(* IEC 61131-3 sources: ae-conveyorline/src, 7 files *)

(* ---- ConveyorSimulation.st ---- *)
USING System.Timer;

NAMESPACE Simatic.Ax.Simulation
    /// Simulation class for conveyor sensor signals using shift register approach
    /// Simulates packages moving along 1 conveyor line (3 conveyors total)
    CLASS ConveyorSimulation
        VAR CONSTANT
            CONVEYOR_LENGTH : LREAL := 2.0; // Conveyor length in meters
            CONVEYOR_SPEED : LREAL := 1.5;  // Conveyor speed in m/s
            SHIFT_INTERVAL : TIME := T#100ms; // Time interval for shift register update
            REGISTER_SIZE : INT := 30; // Size of shift register (3 seconds / 100ms = 30 positions)
            PACKAGE_INTERVAL_POSITIONS : INT := 20; // Positions between packages (2s / 100ms = 20)
        END_VAR

        VAR PUBLIC
            /// Enable/disable simulation
            SimulationEnabled : BOOL := FALSE;

            /// Simulated sensor outputs (3 Conveyors)
            Sensor1 : BOOL := FALSE;
            Sensor2 : BOOL := FALSE;
            Sensor3 : BOOL := FALSE;
        END_VAR

        VAR PRIVATE
            // Shift register for the conveyor line
            _shiftRegister : ARRAY[0..29] OF BOOL;

            // Timer for shift register update
            _shiftTimer : OnDelay;
            _shiftTimerReset : BOOL := FALSE;

            // Package generation counter
            _packageCounter : INT := 0;

            // Sensor position mapping (in shift register positions)
            _sensor1Position : INT := 0;   // Position 0 (start)
            _sensor2Position : INT := 10;  // Position 10 (after 1.0s)
            _sensor3Position : INT := 20;  // Position 20 (after 2.0s)

            // Sensor trigger window
            _sensorWindow : INT := 5; // 5 positions = 500ms

            // Initialization flag
            _initialized : BOOL := FALSE;
        END_VAR

        /// Initialize simulation
        METHOD PUBLIC Initialize
            VAR_TEMP
                i : INT;
            END_VAR

            // Clear shift register
            FOR i := 0 TO (REGISTER_SIZE - 1) DO
                _shiftRegister[i] := FALSE;
            END_FOR;

            _packageCounter := 0;
            _initialized := TRUE;
        END_METHOD

        /// Cyclic update method - must be called every PLC cycle
        METHOD PUBLIC Update
            VAR_TEMP
                i : INT;
            END_VAR

            // If simulation is disabled, reset all sensors
            IF NOT SimulationEnabled THEN
                IF _initialized THEN
                    THIS.Initialize();
                    _initialized := FALSE;
                END_IF;
                THIS.ResetAllSensors();
                RETURN;
            END_IF;

            // Initialize on first run
            IF NOT _initialized THEN
                THIS.Initialize();
            END_IF;

            // Update shift register at defined interval
            _shiftTimer(signal := NOT _shiftTimerReset, duration := SHIFT_INTERVAL);

            IF _shiftTimer.output THEN
                // Shift all positions one step forward
                FOR i := (REGISTER_SIZE - 1) TO 1 BY -1 DO
                    _shiftRegister[i] := _shiftRegister[i - 1];
                END_FOR;

                // Generate new packages
                _packageCounter := _packageCounter + 1;
                IF _packageCounter >= PACKAGE_INTERVAL_POSITIONS THEN
                    _shiftRegister[0] := TRUE;
                    _packageCounter := 0;
                ELSE
                    _shiftRegister[0] := FALSE;
                END_IF;

                // Reset timer for next cycle
                _shiftTimerReset := TRUE;
            ELSE
                _shiftTimerReset := FALSE;
            END_IF;

            // Update sensor outputs (3 Conveyors)
            Sensor1 := THIS.CheckSensorWindow(_sensor1Position);
            Sensor2 := THIS.CheckSensorWindow(_sensor2Position);
            Sensor3 := THIS.CheckSensorWindow(_sensor3Position);
        END_METHOD

        /// Reset all sensor outputs
        METHOD PRIVATE ResetAllSensors
            Sensor1 := FALSE;
            Sensor2 := FALSE;
            Sensor3 := FALSE;
        END_METHOD

        /// Check if any position within sensor window contains a package
        METHOD PRIVATE CheckSensorWindow : BOOL
            VAR_INPUT
                centerPosition : INT;
            END_VAR
            VAR_TEMP
                i : INT;
                startPos : INT;
                endPos : INT;
                packageDetected : BOOL := FALSE;
            END_VAR

            // Calculate window range
            startPos := centerPosition;
            endPos := centerPosition + _sensorWindow - 1;

            // Check if any position in window has a package
            FOR i := startPos TO endPos DO
                IF i >= 0 AND i < REGISTER_SIZE THEN
                    IF _shiftRegister[i] THEN
                        packageDetected := TRUE;
                    END_IF;
                END_IF;
            END_FOR;

            CheckSensorWindow := packageDetected;
        END_METHOD

        /// Get shift register state for debugging (returns position value)
        METHOD PUBLIC GetRegisterState : BOOL
            VAR_INPUT
                position : INT;
            END_VAR

            IF position >= 0 AND position < REGISTER_SIZE THEN
                GetRegisterState := _shiftRegister[position];
            ELSE
                GetRegisterState := FALSE;
            END_IF;
        END_METHOD

    END_CLASS
END_NAMESPACE

(* ---- CycleTimeMeasurement.st ---- *)
USING Siemens.Simatic.Clocks;
USING System.Timer;

NAMESPACE Simatic.Ax.Measurement
    /// Class for measuring and averaging PLC cycle time over a configurable period
    CLASS CycleTimeMeasurement
        VAR CONSTANT
            DEFAULT_AVERAGING_PERIOD : TIME := T#1s; // Default 1 second averaging
        END_VAR

        VAR PUBLIC
            /// Current cycle time in milliseconds
            CycleTimeMs : LREAL := 0.0;

            /// Average cycle time over the averaging period (in milliseconds)
            AverageMs : LREAL := 0.0;

            /// Minimum cycle time in the current averaging period (in milliseconds)
            MinMs : LREAL := 999999.0;

            /// Maximum cycle time in the current averaging period (in milliseconds)
            MaxMs : LREAL := 0.0;

            /// Current cycle time in seconds
            CycleTimeSec : LREAL := 0.0;

            /// Number of cycles in current averaging period
            CycleCount : INT := 0;
        END_VAR

        VAR PRIVATE
            // Runtime measurement instance
            _runtimeMeasurement : RuntimeMeasurement;

            // Cycle time data
            _cycleTime : LTIME;
            _cycleTimeNs : LINT;

            // Average calculation
            _cycleTimeSum : LREAL := 0.0;
            _averageTimer : OnDelay;
            _averagingPeriod : TIME := DEFAULT_AVERAGING_PERIOD;

            // Initialization flag
            _initialized : BOOL := FALSE;
        END_VAR

        /// Initialize the measurement with optional custom averaging period
        METHOD PUBLIC Initialize
            VAR_INPUT
                averagingPeriod : TIME := T#1s; // Averaging period (default 1 second)
            END_VAR

            _averagingPeriod := averagingPeriod;
            THIS.Reset();
            _initialized := TRUE;
        END_METHOD

        /// Start measurement at the beginning of the cycle
        METHOD PUBLIC StartCycle
            IF NOT _initialized THEN
                THIS.Initialize();
            END_IF;

            _runtimeMeasurement.Start();
        END_METHOD

        /// Stop measurement at the end of the cycle and calculate statistics
        METHOD PUBLIC StopCycle
            // Stop runtime measurement and get cycle time
            _cycleTime := _runtimeMeasurement.Stop();

            // Get elapsed time in different formats
            _cycleTimeNs := _runtimeMeasurement.GetElapsedNanoseconds();
            CycleTimeSec := _runtimeMeasurement.GetElapsedSeconds();

            // Convert nanoseconds to milliseconds for easier reading
            CycleTimeMs := TO_LREAL(_cycleTimeNs) / 1000000.0;

            // Calculate average over the configured period
            _cycleTimeSum := _cycleTimeSum + CycleTimeMs;
            CycleCount := CycleCount + 1;

            // Track min/max
            IF CycleTimeMs < MinMs THEN
                MinMs := CycleTimeMs;
            END_IF;
            IF CycleTimeMs > MaxMs THEN
                MaxMs := CycleTimeMs;
            END_IF;

            // Check if averaging period has elapsed
            _averageTimer(signal := TRUE, duration := _averagingPeriod);

            IF _averageTimer.output THEN
                // Calculate average
                IF CycleCount > 0 THEN
                    AverageMs := _cycleTimeSum / TO_LREAL(CycleCount);
                END_IF;

                // Reset for next averaging period
                _cycleTimeSum := 0.0;
                CycleCount := 0;
                MinMs := 999999.0;
                MaxMs := 0.0;
                _averageTimer(signal := FALSE, duration := _averagingPeriod);
            END_IF;
        END_METHOD

        /// Reset all measurements
        METHOD PUBLIC Reset
            _cycleTimeSum := 0.0;
            CycleCount := 0;
            MinMs := 999999.0;
            MaxMs := 0.0;
            CycleTimeMs := 0.0;
            AverageMs := 0.0;
            CycleTimeSec := 0.0;
            _averageTimer(signal := FALSE, duration := _averagingPeriod);
        END_METHOD

        /// Get the current cycle time in nanoseconds
        METHOD PUBLIC GetCycleTimeNs : LINT
            GetCycleTimeNs := _cycleTimeNs;
        END_METHOD

        /// Get the raw LTIME value
        METHOD PUBLIC GetCycleTime : LTIME
            GetCycleTime := _cycleTime;
        END_METHOD

    END_CLASS
END_NAMESPACE

(* ---- SimpleRelease.st ---- *)
USING Simatic.Ax.AutomationBase;

NAMESPACE Simatic.Ax.Conveyor

    /// Simple release implementation that can be controlled by a boolean signal
    /// Used to enable/disable equipment operation (e.g., safety interlocks, enable signals)
    CLASS SimpleRelease IMPLEMENTS IRelease
        VAR PUBLIC
            /// Release signal - TRUE allows operation, FALSE prevents operation
            Signal : BOOL := TRUE;
        END_VAR

        /// Returns TRUE when equipment is released and allowed to operate
        METHOD PUBLIC IsReleased : BOOL
            IsReleased := Signal;
        END_METHOD
    END_CLASS

END_NAMESPACE

(* ---- Configuration.st ---- *)
USING Simatic.Ax.Conveyor;
USING Simatic.Ax.IO.Input;
USING Simatic.Ax.IO.Output;
USING Simatic.Ax.Motor;
USING Simatic.Ax.AutomationBase;
USING Simatic.Ax.Simulation;

CONFIGURATION MyConfiguration
    TASK Main (PRIORITY := 1);
    PROGRAM P0 WITH Main : HardwareInputs;
    PROGRAM P1 WITH Main : MainProgram;
    PROGRAM P2 WITH Main : HardwareOutputs;
    VAR_GLOBAL
        // Manual Mode
        ManualMode : BOOL := FALSE;

        // Reset button for all conveyors (BinSignal from @simatic-ax/io)
        ResetButton : BinSignal;

        // Conveyor simulation for sensor signals
        ConveyorSim : ConveyorSimulation;

        // Global operating mode manager (shared by all conveyors)
        GlobalOpMode : OperatingModeManager;

        // Global reset command manager (shared by all conveyors)
        GlobalResetManager : ResetCommandManager := (ResetSignal := ResetButton);

        // Global release signal (shared by all conveyors)
        GlobalRelease : SimpleRelease := (Signal := TRUE);

        // Motor outputs using BinOutput (3 Conveyors)
        MotorOutput1 : BinOutput;
        MotorOutput2 : BinOutput;
        MotorOutput3 : BinOutput;

        // Motors for each conveyor (3 Conveyors)
        Motor1 : MotorGeneric := (MotorOutput := MotorOutput1, ExternalRelease := GlobalRelease);
        Motor2 : MotorGeneric := (MotorOutput := MotorOutput2, ExternalRelease := GlobalRelease);
        Motor3 : MotorGeneric := (MotorOutput := MotorOutput3, ExternalRelease := GlobalRelease);

        // Stop sensors (3 Conveyors)
        StopSensor1 : BinSignal;
        StopSensor2 : BinSignal;
        StopSensor3 : BinSignal;

        // Conveyor line (3 Conveyors in series)
        Conveyor1 : ConveyorBase := (
            Name := 'Conveyor_1',
            StopSensor := StopSensor1,
            Motor := Motor1,
            NextConveyor := Conveyor2,
            PrevConveyor := NULL,
            OffDelayTime := T#5s,
            Mode := GlobalOpMode,
            ExternalRelease := GlobalRelease,
            ResetCommand := GlobalResetManager);

        Conveyor2 : ConveyorBase := (
            Name := 'Conveyor_2',
            StopSensor := StopSensor2,
            Motor := Motor2,
            NextConveyor := Conveyor3,
            PrevConveyor := Conveyor1,
            OffDelayTime := T#5s,
            Mode := GlobalOpMode,
            ExternalRelease := GlobalRelease,
            ResetCommand := GlobalResetManager);

        Conveyor3 : ConveyorBase := (
            Name := 'Conveyor_3',
            StopSensor := StopSensor3,
            Motor := Motor3,
            NextConveyor := NULL,
            PrevConveyor := Conveyor2,
            OffDelayTime := T#5s,
            Mode := GlobalOpMode,
            ExternalRelease := GlobalRelease,
            ResetCommand := GlobalResetManager);

        // Physical I/O mapping (3 Conveyors)
        HW_StopSensor1 AT %I0.0 : BOOL;
        HW_StopSensor2 AT %I0.1 : BOOL;
        HW_StopSensor3 AT %I0.2 : BOOL;
        // Motor outputs (3 Conveyors)
        HW_Motor1_Run AT %Q0.0 : BOOL;
        HW_Motor2_Run AT %Q0.1 : BOOL;
        HW_Motor3_Run AT %Q0.2 : BOOL;
        // Physical I/O for Reset Button
        HW_ResetButton AT %I0.3 : BOOL;
    END_VAR
END_CONFIGURATION

(* ---- InputProgram.st ---- *)
USING Simatic.Ax.IO.Input;
USING Simatic.Ax.Simulation;

PROGRAM HardwareInputs
    VAR_EXTERNAL
        // Reset button for all conveyors (BinSignal)
        ResetButton : BinSignal;

        // Stop sensors (3 Conveyors)
        StopSensor1 : BinSignal;
        StopSensor2 : BinSignal;
        StopSensor3 : BinSignal;

        // Conveyor simulation
        ConveyorSim : ConveyorSimulation;

        // Physical I/O (3 Conveyors)
        HW_StopSensor1 : BOOL;
        HW_StopSensor2 : BOOL;
        HW_StopSensor3 : BOOL;

        // Physical I/O for Reset Button
        HW_ResetButton : BOOL;
    END_VAR

    VAR
        EffectiveStopSensor1 : BOOL := FALSE;
        EffectiveStopSensor2 : BOOL := FALSE;
        EffectiveStopSensor3 : BOOL := FALSE;
    END_VAR

    // Read reset button input
    ResetButton.ReadCyclic(signal := HW_ResetButton);

    // If simulation is enabled, use simulated sensor values
    // If simulation is disabled, reset all sensor signals to FALSE
    IF ConveyorSim.SimulationEnabled THEN
        EffectiveStopSensor1 := ConveyorSim.Sensor1;
        EffectiveStopSensor2 := ConveyorSim.Sensor2;
        EffectiveStopSensor3 := ConveyorSim.Sensor3;
    ELSE
        EffectiveStopSensor1 := HW_StopSensor1;
        EffectiveStopSensor2 := HW_StopSensor2;
        EffectiveStopSensor3 := HW_StopSensor3;
    END_IF;

    // Read physical inputs and update BinSignals (3 Conveyors)
    StopSensor1.ReadCyclic(signal := EffectiveStopSensor1);
    StopSensor2.ReadCyclic(signal := EffectiveStopSensor2);
    StopSensor3.ReadCyclic(signal := EffectiveStopSensor3);
END_PROGRAM

(* ---- MainProgram.st ---- *)
USING Simatic.Ax.Conveyor;
USING Simatic.Ax.Motor;
USING Simatic.Ax.AutomationBase;
USING Simatic.Ax.Simulation;
USING Simatic.Ax.Measurement;
USING System.Timer;

PROGRAM MainProgram
    VAR_EXTERNAL

        // Manual Mode
        ManualMode : BOOL;

        // Conveyor line (3 Conveyors)
        Conveyor1 : ConveyorBase;
        Conveyor2 : ConveyorBase;
        Conveyor3 : ConveyorBase;

        // Global operating mode manager (shared by all conveyors)
        GlobalOpMode : OperatingModeManager;

        // Global reset command manager (shared by all conveyors)
        GlobalResetManager : ResetCommandManager;

        // Global release signal (shared by all conveyors)
        GlobalRelease : SimpleRelease;

        // Conveyor simulation
        ConveyorSim : ConveyorSimulation;

    END_VAR

    VAR
        // Cycle time measurement (encapsulated)
        _cycleTimeMeasurement : CycleTimeMeasurement;

        // Current and average cycle time values
        CurrentCycleTimeMs : LREAL := 0.0;
        AverageCycleTimeMs : LREAL := 0.0;
    END_VAR

    VAR_TEMP
    END_VAR

    // Start cycle time measurement
    _cycleTimeMeasurement.StartCycle();

    // Handle operating mode
    IF ManualMode THEN
        GlobalOpMode.SetOperatingMode(mode := OperatingModes#Manual);
    ELSE
        GlobalOpMode.SetOperatingMode(mode := OperatingModes#Automatic);
    END_IF;

    // ========================================
    // CYCLIC EXECUTION - Called every PLC cycle
    // ========================================

    // 0. Update simulation (if enabled, overwrites HW inputs)
    ConveyorSim.Update();

    // 1. Execute conveyor logic (3 Conveyors)
    Conveyor1.RunCyclic();
    Conveyor2.RunCyclic();
    Conveyor3.RunCyclic();

    // 2. Execute reset manager cyclic (MUST be called after all equipment)
    GlobalResetManager.RunCyclic();

    // Stop cycle time measurement and calculate statistics
    _cycleTimeMeasurement.StopCycle();

    // Assign values to local variables
    CurrentCycleTimeMs := _cycleTimeMeasurement.CycleTimeMs;
    AverageCycleTimeMs := _cycleTimeMeasurement.AverageMs;

END_PROGRAM

(* ---- OutputProgram.st ---- *)
USING Simatic.Ax.IO.Output;

PROGRAM HardwareOutputs
    VAR_EXTERNAL
        // Motor outputs (3 Conveyors)
        MotorOutput1 : BinOutput;
        MotorOutput2 : BinOutput;
        MotorOutput3 : BinOutput;

        // Physical I/O - Motors (3 Conveyors)
        HW_Motor1_Run : BOOL;
        HW_Motor2_Run : BOOL;
        HW_Motor3_Run : BOOL;
    END_VAR

    // Write motor states to physical outputs (3 Conveyors)
    MotorOutput1.WriteCyclic(Q => HW_Motor1_Run);
    MotorOutput2.WriteCyclic(Q => HW_Motor2_Run);
    MotorOutput3.WriteCyclic(Q => HW_Motor3_Run);
END_PROGRAM
